% RSLogix 500 project SEND_DATA_2.RSS, saved by version 8.10.00.18 %
PROJECT "UNTITLED"    % processor: Bul.1763 MicroLogix 1100 Series B %

PROGRAM FILES
  LAD 2 "MAIN"  5 rungs
  LAD 3 "CLOCK"  19 rungs
  LAD 4 "SEND"  7 rungs  % COMMUNICATION %
  LAD 6 "START I2C"  5 rungs
  LAD 5: only END

DATA FILES
  O0 OUTPUT  4 elements
  I1 INPUT  6 elements
  S2 STATUS  66 elements
  B3 BINARY  1 elements
  T4 TIMER  4 elements
  C5 COUNTER  3 elements
  R6 CONTROL  1 elements
  N7 INTEGER  13 elements
  F8 FLOAT  1 elements

LADDER 2 "MAIN"
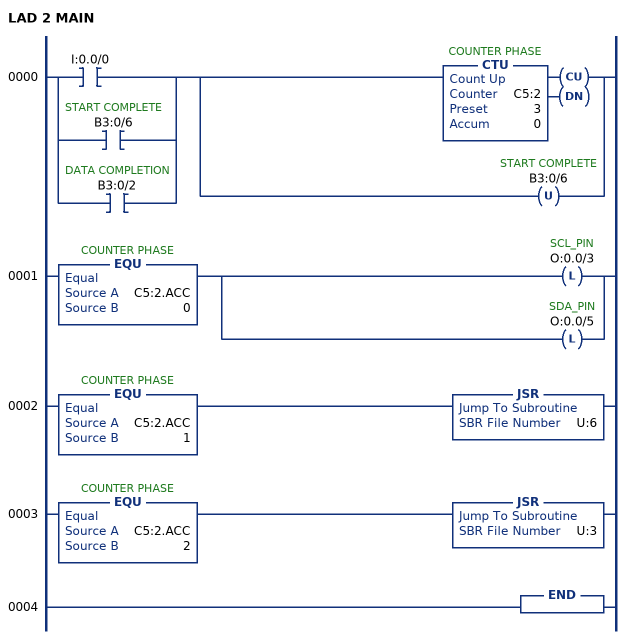
% Rung: 0 %
SOR BST XIC I:0.0/0 NXB BST XIC B3:0/6 NXB XIC B3:0/2 BND BND BST CTU C5:2 3 0 NXB OTU B3:0/6 BND EOR
%   XIC I:0.0/0  "send_data" %
%   B3:0/6  "START COMPLETE" %
%   B3:0/2  "DATA COMPLETION" %
%   C5:2  "COUNTER PHASE" %
% Rung: 1 %
SOR EQU C5:2.ACC 0 BST OTL O:0.0/3 NXB OTL O:0.0/5 BND EOR
%   C5:2  "COUNTER PHASE" %
%   O:0.0/3  "SCL_PIN" %
%   O:0.0/5  "SDA_PIN" %
% Rung: 2 %
SOR EQU C5:2.ACC 1 JSR U:6 EOR
%   C5:2  "COUNTER PHASE" %
% Rung: 3 %
SOR EQU C5:2.ACC 2 JSR U:3 EOR
%   C5:2  "COUNTER PHASE" %
% Rung: 4 %
SOR END EOR

LADDER 3 "CLOCK"
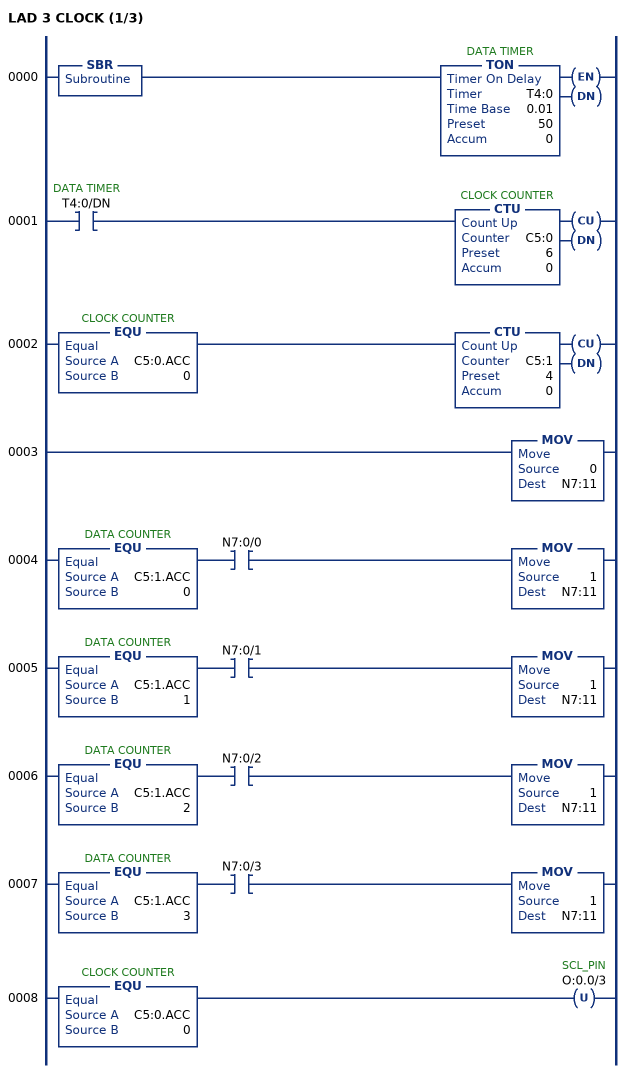
% Rung: 0 %
SOR SBR TON T4:0 0.01 50 0 EOR
%   T4:0  "DATA TIMER" %
% Rung: 1 %
SOR XIC T4:0/DN CTU C5:0 6 0 EOR
%   T4:0  "DATA TIMER" %
%   C5:0  "CLOCK COUNTER" %
% Rung: 2 %
SOR EQU C5:0.ACC 0 CTU C5:1 4 0 EOR
%   C5:0  "CLOCK COUNTER" %
% Rung: 3 %
SOR MOV 0 N7:11 EOR
% Rung: 4 %
SOR EQU C5:1.ACC 0 XIC N7:0/0 MOV 1 N7:11 EOR
%   C5:1.ACC  "DATA COUNTER" %
% Rung: 5 %
SOR EQU C5:1.ACC 1 XIC N7:0/1 MOV 1 N7:11 EOR
%   C5:1.ACC  "DATA COUNTER" %
% Rung: 6 %
SOR EQU C5:1.ACC 2 XIC N7:0/2 MOV 1 N7:11 EOR
%   C5:1.ACC  "DATA COUNTER" %
% Rung: 7 %
SOR EQU C5:1.ACC 3 XIC N7:0/3 MOV 1 N7:11 EOR
%   C5:1.ACC  "DATA COUNTER" %
% Rung: 8 %
SOR EQU C5:0.ACC 0 OTU O:0.0/3 EOR
%   C5:0  "CLOCK COUNTER" %
%   O:0.0/3  "SCL_PIN" %

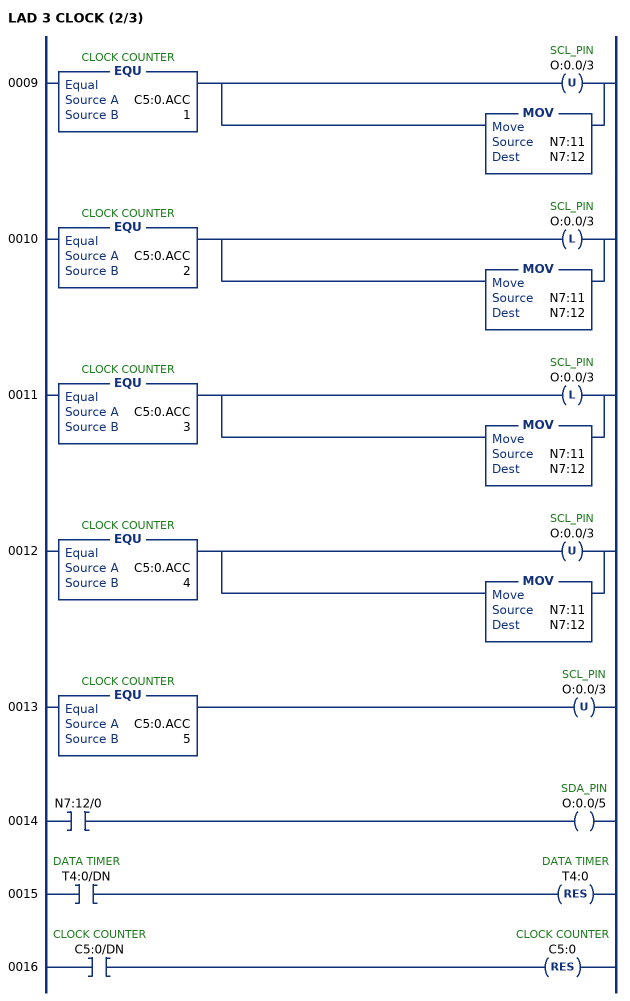
% Rung: 9 %
SOR EQU C5:0.ACC 1 BST OTU O:0.0/3 NXB MOV N7:11 N7:12 BND EOR
%   C5:0  "CLOCK COUNTER" %
%   O:0.0/3  "SCL_PIN" %
% Rung: 10 %
SOR EQU C5:0.ACC 2 BST OTL O:0.0/3 NXB MOV N7:11 N7:12 BND EOR
%   C5:0  "CLOCK COUNTER" %
%   O:0.0/3  "SCL_PIN" %
% Rung: 11 %
SOR EQU C5:0.ACC 3 BST OTL O:0.0/3 NXB MOV N7:11 N7:12 BND EOR
%   C5:0  "CLOCK COUNTER" %
%   O:0.0/3  "SCL_PIN" %
% Rung: 12 %
SOR EQU C5:0.ACC 4 BST OTU O:0.0/3 NXB MOV N7:11 N7:12 BND EOR
%   C5:0  "CLOCK COUNTER" %
%   O:0.0/3  "SCL_PIN" %
% Rung: 13 %
SOR EQU C5:0.ACC 5 OTU O:0.0/3 EOR
%   C5:0  "CLOCK COUNTER" %
%   O:0.0/3  "SCL_PIN" %
% Rung: 14 %
SOR XIC N7:12/0 OTE O:0.0/5 EOR
%   O:0.0/5  "SDA_PIN" %
% Rung: 15 %
SOR XIC T4:0/DN RES T4:0 EOR
%   T4:0  "DATA TIMER" %
% Rung: 16 %
SOR XIC C5:0/DN RES C5:0 EOR
%   C5:0  "CLOCK COUNTER" %

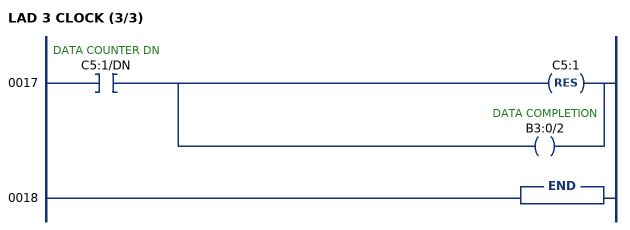
% Rung: 17 %
SOR XIC C5:1/DN BST RES C5:1 NXB OTE B3:0/2 BND EOR
%   C5:1/DN  "DATA COUNTER DN" %
%   B3:0/2  "DATA COMPLETION" %
% Rung: 18 %
SOR END EOR

LADDER 4 "SEND"    % COMMUNICATION %
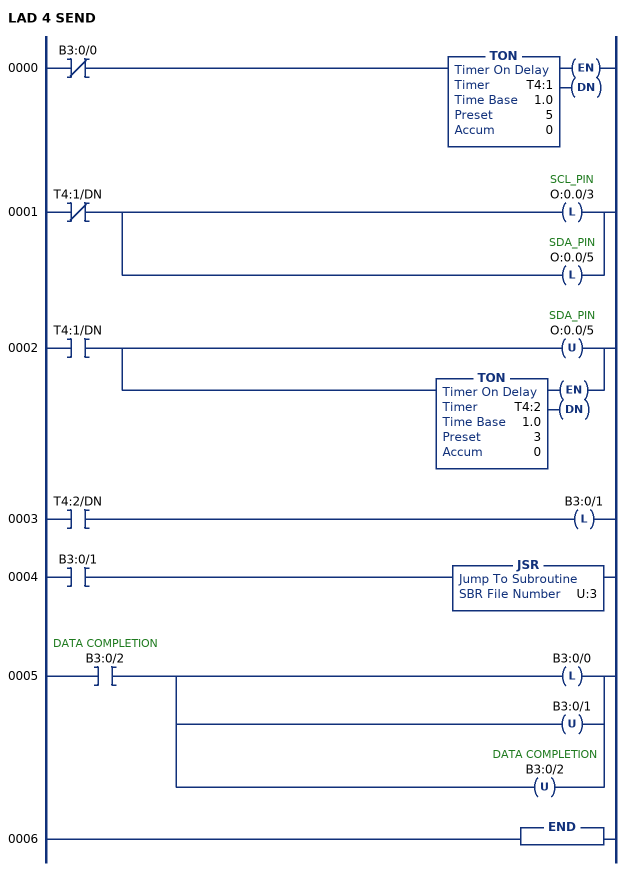
% Rung: 0 %
SOR XIO B3:0/0 TON T4:1 1.0 5 0 EOR
%   TON T4:1  "INIT TIMER" %
% Rung: 1 %
SOR XIO T4:1/DN BST OTL O:0.0/3 NXB OTL O:0.0/5 BND EOR
%   O:0.0/3  "SCL_PIN" %
%   O:0.0/5  "SDA_PIN" %
% Rung: 2 %
SOR XIC T4:1/DN BST OTU O:0.0/5 NXB TON T4:2 1.0 3 0 BND EOR
%   XIC T4:1/DN  "timer_reached" %
%   O:0.0/5  "SDA_PIN" %
% Rung: 3 %
SOR XIC T4:2/DN OTL B3:0/1 EOR
% Rung: 4 %
SOR XIC B3:0/1 JSR U:3 EOR
% Rung: 5 %
SOR XIC B3:0/2 BST OTL B3:0/0 NXB BST OTU B3:0/1 NXB OTU B3:0/2 BND BND EOR
%   B3:0/2  "DATA COMPLETION" %
% Rung: 6 %
SOR END EOR

LADDER 6 "START I2C"
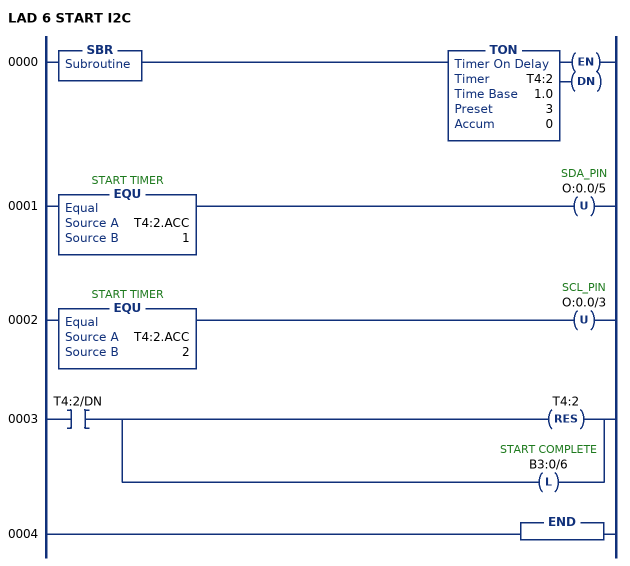
% Rung: 0 %
SOR SBR TON T4:2 1.0 3 0 EOR
% Rung: 1 %
SOR EQU T4:2.ACC 1 OTU O:0.0/5 EOR
%   T4:2.ACC  "START TIMER" %
%   O:0.0/5  "SDA_PIN" %
% Rung: 2 %
SOR EQU T4:2.ACC 2 OTU O:0.0/3 EOR
%   T4:2.ACC  "START TIMER" %
%   O:0.0/3  "SCL_PIN" %
% Rung: 3 %
SOR XIC T4:2/DN BST RES T4:2 NXB OTL B3:0/6 BND EOR
%   B3:0/6  "START COMPLETE" %
% Rung: 4 %
SOR END EOR

OTHER DOCUMENTED ADDRESSES
  B3:0/4  "STOP INIT I2c"
  B3:0/5  "SENDING START"
  B3:0/7  "START DATA"
  N7:10  "CLOCK VARIABLE"
  O:0.0/1  "SCL"
  U3  

DATA TABLE (non-zero values as saved)
DATA T4
% .PRE .ACC %
% T4:0 % 50 0
% T4:1 % 5 0
% T4:2 % 3 0
% T4:3 % 10 0
DATA C5
% .PRE .ACC %
% C5:0 % 6 0
% C5:1 % 4 0
% C5:2 % 3 0
DATA N7
% N7:0 % 5 0 0 0 0 0 0 0 0 0
